Staubli VAL3: type2.pjx

--- type2.pjx ---
Parameters version=s7.6.3 stackSize=5000 millimeterUnit=true
Data file=type2.dtx
Type name=TrajBigBox path=Disk://goHome/template/TrajBigBox/TrajBigBox.pjx

--- type2.dtx ---
public TrajBigBox box{}
